FUNCTION_BLOCK Test_FormatStringWith4CharHexValue EXTENDS TUnitTestBase
VAR_INPUT
END_VAR
VAR_OUTPUT
END_VAR
VAR
    FormattedString : T_MaxString;
    Value : UINT;
END_VAR

Value := 16#12AB;
FormattedString := F_FormatString1('Hex value = 0x%0.4X',F_UINT(Value));

Assertion.AssertEquals_STRING(
    Expected     := 'Hex value = 0x12AB', 
    Actual       := FormattedString, 
    ObjectName   := _TestName, 
    VariableName := 'FormattedString');

TestFinished();

END_FUNCTION_BLOCK

(* stored: Version 1.1.0.1, ProductVersion 3.1.4024.3
   POU Test_FormatStringWith4CharHexValue: Id {c0c11d44-c536-4c7d-853a-9e40b1c7fd63}, SpecialFunc None *)
